PROGRAM DemandedSpeedTask
VAR
	{attribute 'UserUnit' := '<AngularVelocity, RPM, RPM, 9.549296596425, 0, 0 >'}
	DemandedSpeed : UINT;
	DemandedSpeedImpl : AnalogPrescaledSpeedCalculator;
END_VAR

DemandedSpeed := DemandedSpeedImpl.GetSpeed();

END_PROGRAM

(* stored: Version 1.1.0.1, ProductVersion 3.1.4022.17
   POU DemandedSpeedTask: Id {2c74394b-eed0-495f-90ea-7d865744d37f}, SpecialFunc None *)
